PROGRAM POU_SM01_LineBend
VAR
END_VAR

IF LineAngle < -LINE_ANGLE_SCALING THEN
	
	R100_01 				:= TRUE;
	
ELSE
	
	R100_01					:= FALSE;
	
END_IF

IF LineAngle > LINE_ANGLE_SCALING THEN
	
	R100_04 				:= TRUE;
	
ELSE
	
	R100_04					:= FALSE;
	
END_IF

END_PROGRAM

(* stored: Version 1.1.0.1, ProductVersion 3.1.4022.7
   POU POU_SM01_LineBend: Id {2189710a-6cb8-4a79-8677-e78bd700b2e9}, SpecialFunc None *)
